// Mitsubishi GX Works2 project: NAND   PLC: Q03UDV

PROGRAM MAIN
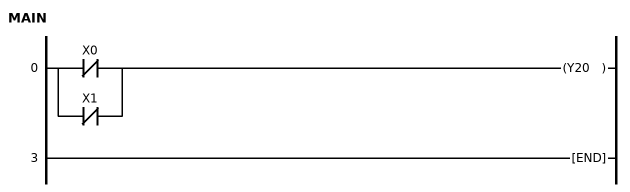
0     LDI     X0
      ORI     X1
      OUT     Y20
3     END
END_PROGRAM
